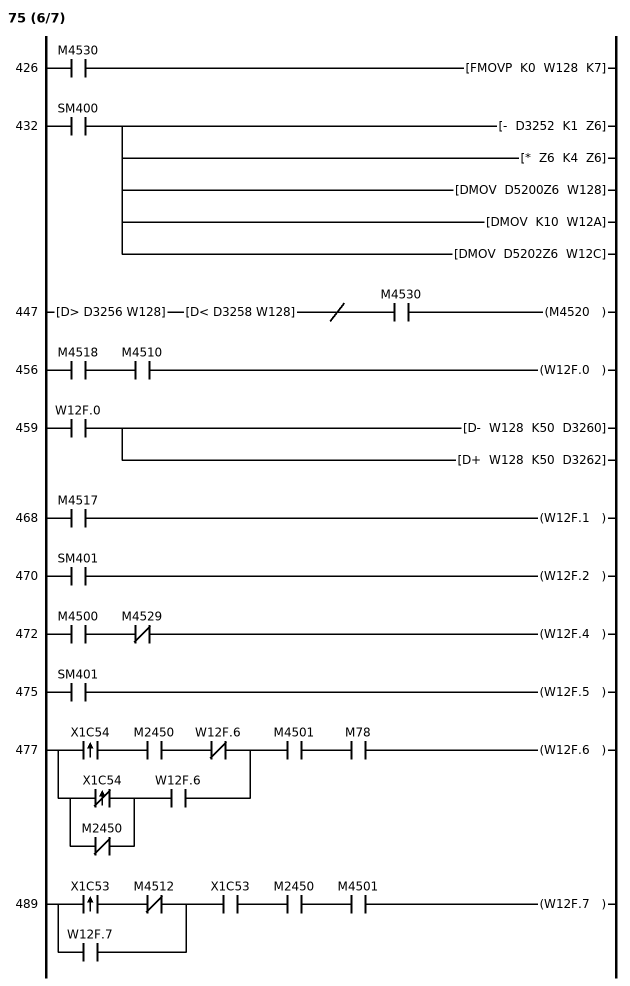
426   LD      M4530
      FMOVP   K0 W128 K7
432   LD      SM400
      -       D3252 K1 Z6
      *       Z6 K4 Z6
      DMOV    D5200Z6 W128
      DMOV    K10 W12A
      DMOV    D5202Z6 W12C
447   LDD>    D3256 W128
      ANDD<   D3258 W128
      INV
      AND     M4530
      OUT     M4520
456   LD      M4518
      AND     M4510
      OUT     W12F.0
459   LD      W12F.0
      D-      W128 K50 D3260
      D+      W128 K50 D3262
468   LD      M4517
      OUT     W12F.1
470   LD      SM401
      OUT     W12F.2
472   LD      M4500
      ANI     M4529
      OUT     W12F.4
475   LD      SM401
      OUT     W12F.5
477   LDP     X1C54
      AND     M2450
      ANI     W12F.6
      LDPI    X1C54
      ORI     M2450
      AND     W12F.6
      ORB
      AND     M4501
      AND     M78
      OUT     W12F.6
489   LDP     X1C53
      ANI     M4512
      OR      W12F.7
      AND     X1C53
      AND     M2450
      AND     M4501
      OUT     W12F.7
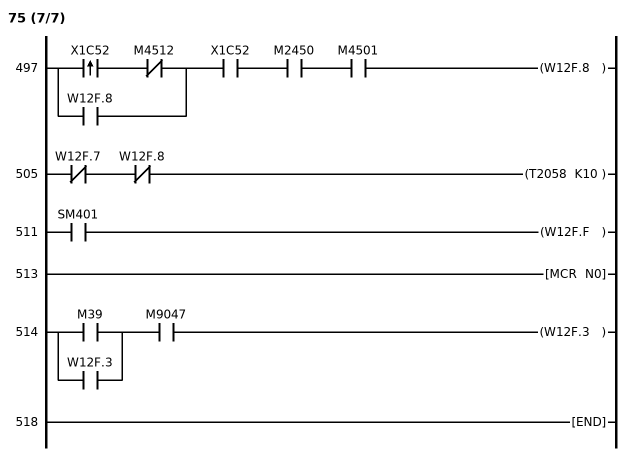
497   LDP     X1C52
      ANI     M4512
      OR      W12F.8
      AND     X1C52
      AND     M2450
      AND     M4501
      OUT     W12F.8
505   LDI     W12F.7
      ANI     W12F.8
      OUT     T2058 K10
511   LD      SM401
      OUT     W12F.F
513   MCR     N0
514   LD      M39
      OR      W12F.3
      AND     M9047
      OUT     W12F.3
518   END
END_PROGRAM

PROGRAM 76
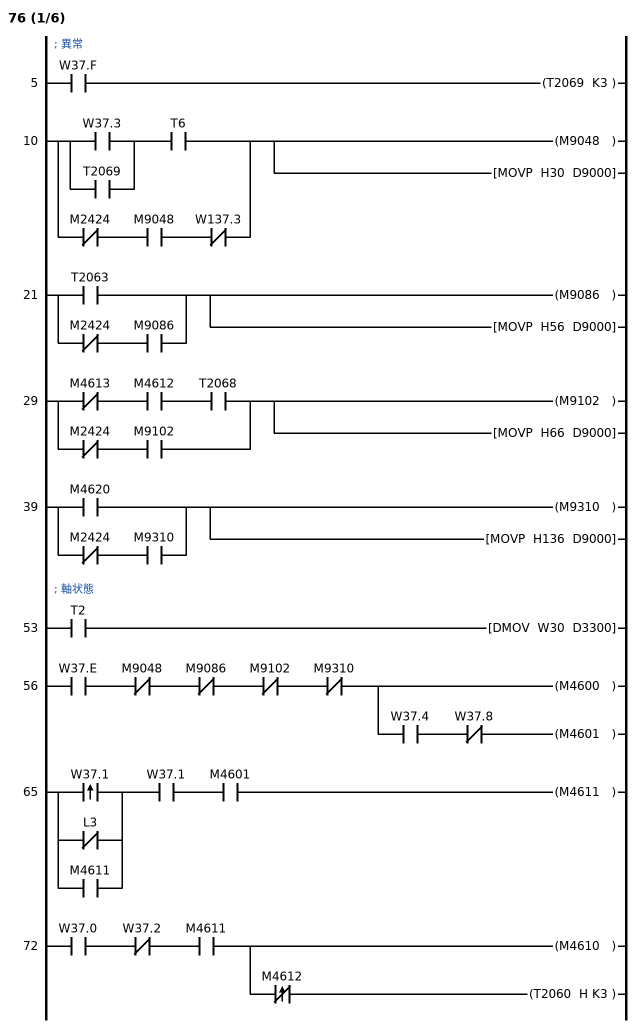
; 異常
5     LD      W37.F
      OUT     T2069 K3
10    LD      W37.3
      OR      T2069
      AND     T6
      LDI     M2424
      AND     M9048
      ANI     W137.3
      ORB
      OUT     M9048
      MOVP    H30 D9000
21    LD      T2063
      LDI     M2424
      AND     M9086
      ORB
      OUT     M9086
      MOVP    H56 D9000
29    LDI     M4613
      AND     M4612
      AND     T2068
      LDI     M2424
      AND     M9102
      ORB
      OUT     M9102
      MOVP    H66 D9000
39    LD      M4620
      LDI     M2424
      AND     M9310
      ORB
      OUT     M9310
      MOVP    H136 D9000
; 軸状態
53    LD      T2
      DMOV    W30 D3300
56    LD      W37.E
      ANI     M9048
      ANI     M9086
      ANI     M9102
      ANI     M9310
      OUT     M4600
      AND     W37.4
      ANI     W37.8
      OUT     M4601
65    LDP     W37.1
      ORI     L3
      OR      M4611
      AND     W37.1
      AND     M4601
      OUT     M4611
72    LD      W37.0
      ANI     W37.2
      AND     M4611
      OUT     M4610
      ANDPI   M4612
      OUTH    T2060 K3
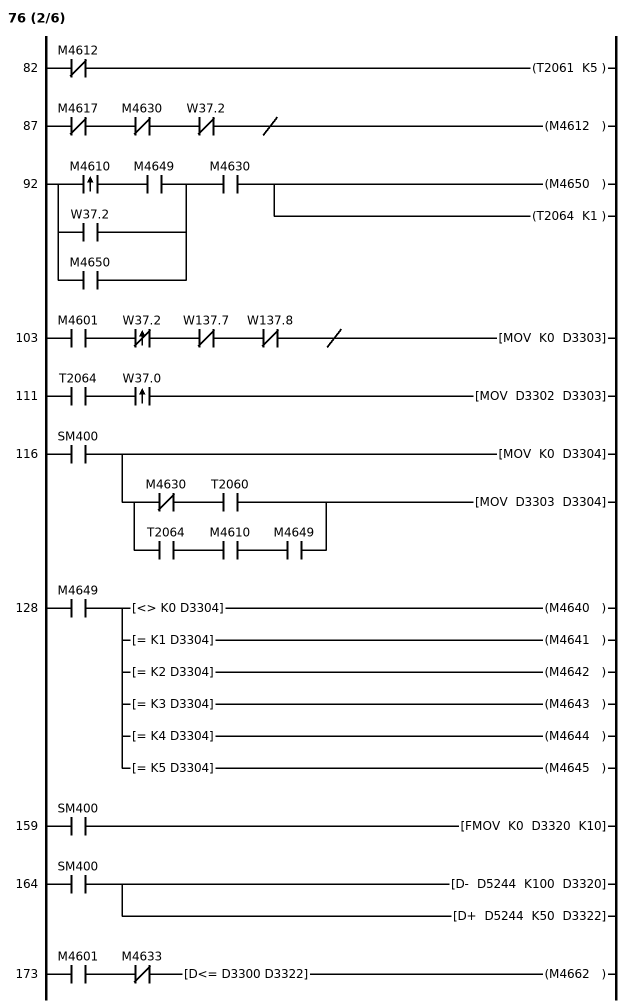
82    LDI     M4612
      OUT     T2061 K5
87    LDI     M4617
      ANI     M4630
      ANI     W37.2
      INV
      OUT     M4612
92    LDP     M4610
      AND     M4649
      OR      W37.2
      OR      M4650
      AND     M4630
      OUT     M4650
      OUT     T2064 K1
103   LD      M4601
      ANDPI   W37.2
      ANI     W137.7
      ANI     W137.8
      INV
      MOV     K0 D3303
111   LD      T2064
      ANDP    W37.0
      MOV     D3302 D3303
116   LD      SM400
      MOV     K0 D3304
      LDI     M4630
      AND     T2060
      LD      T2064
      AND     M4610
      AND     M4649
      ORB
      ANB
      MOV     D3303 D3304
128   LD      M4649
      MPS
      AND<>   K0 D3304
      OUT     M4640
      MRD
      AND=    K1 D3304
      OUT     M4641
      MRD
      AND=    K2 D3304
      OUT     M4642
      MRD
      AND=    K3 D3304
      OUT     M4643
      MRD
      AND=    K4 D3304
      OUT     M4644
      MPP
      AND=    K5 D3304
      OUT     M4645
159   LD      SM400
      FMOV    K0 D3320 K10
164   LD      SM400
      D-      D5244 K100 D3320
      D+      D5244 K50 D3322
173   LD      M4601
      ANI     M4633
      ANDD<=  D3300 D3322
      OUT     M4662
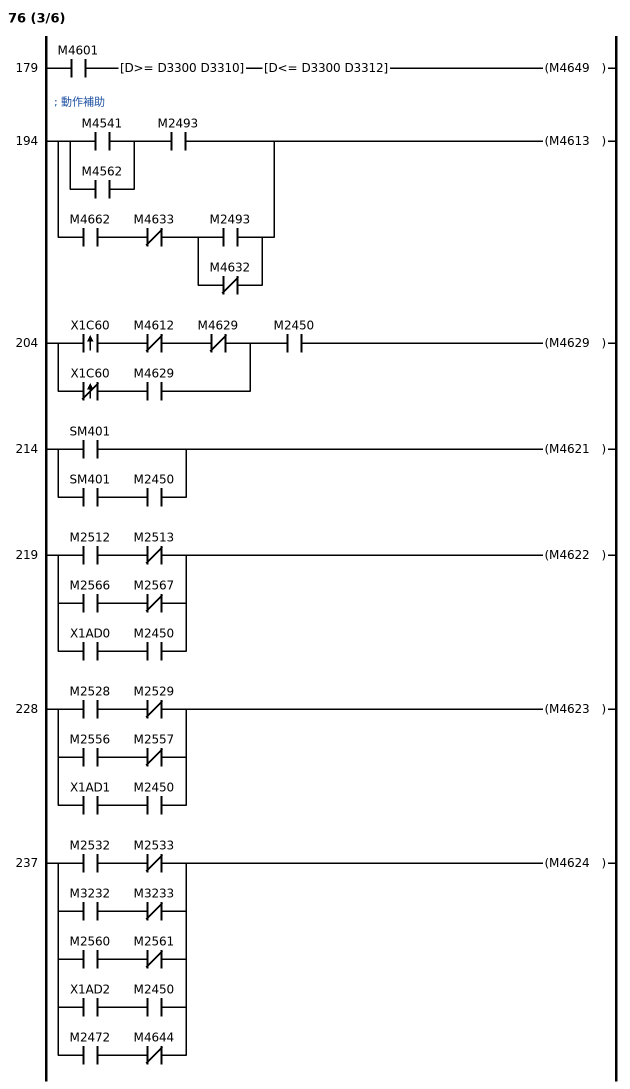
179   LD      M4601
      ANDD>=  D3300 D3310
      ANDD<=  D3300 D3312
      OUT     M4649
; 動作補助
194   LD      M4541
      OR      M4562
      AND     M2493
      LD      M4662
      ANI     M4633
      LD      M2493
      ORI     M4632
      ANB
      ORB
      OUT     M4613
204   LDP     X1C60
      ANI     M4612
      ANI     M4629
      LDPI    X1C60
      AND     M4629
      ORB
      AND     M2450
      OUT     M4629
214   LD      SM401
      LD      SM401
      AND     M2450
      ORB
      OUT     M4621
219   LD      M2512
      ANI     M2513
      LD      M2566
      ANI     M2567
      ORB
      LD      X1AD0
      AND     M2450
      ORB
      OUT     M4622
228   LD      M2528
      ANI     M2529
      LD      M2556
      ANI     M2557
      ORB
      LD      X1AD1
      AND     M2450
      ORB
      OUT     M4623
237   LD      M2532
      ANI     M2533
      LD      M3232
      ANI     M3233
      ORB
      LD      M2560
      ANI     M2561
      ORB
      LD      X1AD2
      AND     M2450
      ORB
      LD      M2472
      ANI     M4644
      ORB
      OUT     M4624
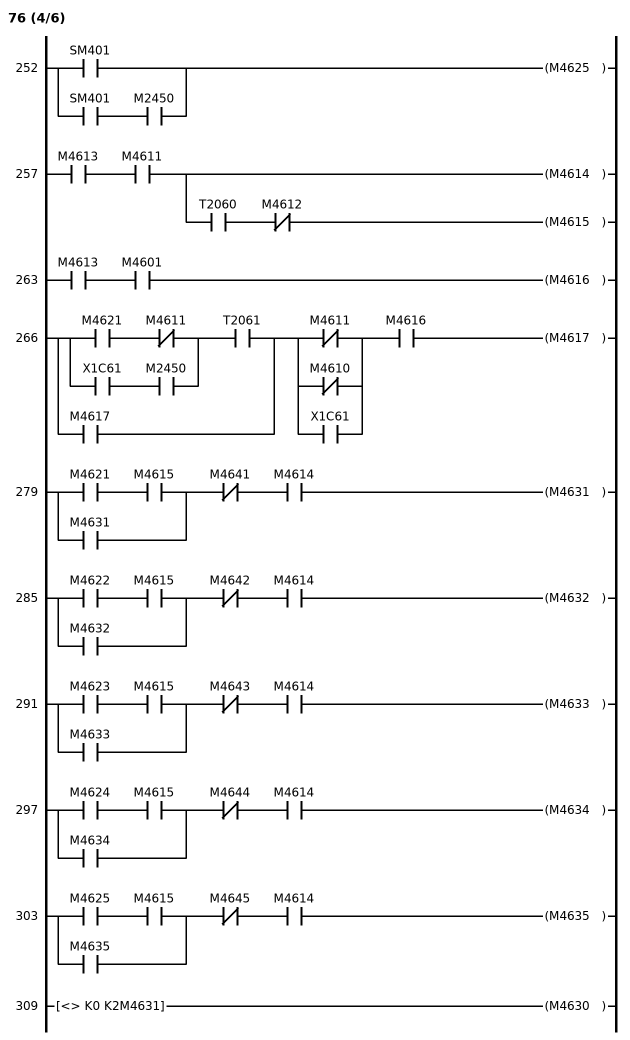
252   LD      SM401
      LD      SM401
      AND     M2450
      ORB
      OUT     M4625
257   LD      M4613
      AND     M4611
      OUT     M4614
      AND     T2060
      ANI     M4612
      OUT     M4615
263   LD      M4613
      AND     M4601
      OUT     M4616
266   LD      M4621
      ANI     M4611
      LD      X1C61
      AND     M2450
      ORB
      AND     T2061
      OR      M4617
      LDI     M4611
      ORI     M4610
      OR      X1C61
      ANB
      AND     M4616
      OUT     M4617
279   LD      M4621
      AND     M4615
      OR      M4631
      ANI     M4641
      AND     M4614
      OUT     M4631
285   LD      M4622
      AND     M4615
      OR      M4632
      ANI     M4642
      AND     M4614
      OUT     M4632
291   LD      M4623
      AND     M4615
      OR      M4633
      ANI     M4643
      AND     M4614
      OUT     M4633
297   LD      M4624
      AND     M4615
      OR      M4634
      ANI     M4644
      AND     M4614
      OUT     M4634
303   LD      M4625
      AND     M4615
      OR      M4635
      ANI     M4645
      AND     M4614
      OUT     M4635
309   LD<>    K0 K2M4631
      OUT     M4630
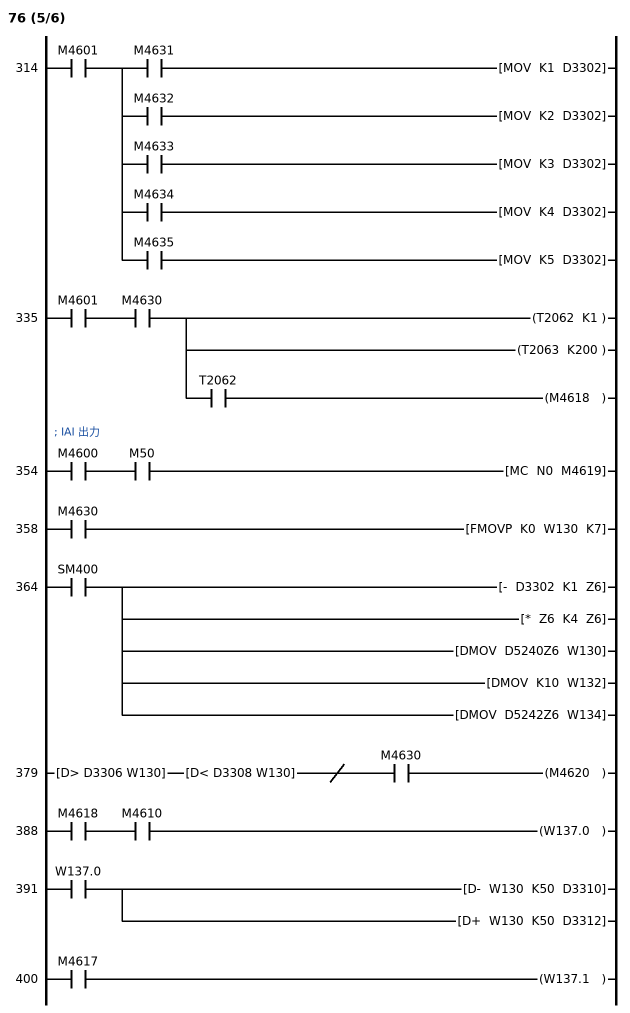
314   LD      M4601
      MPS
      AND     M4631
      MOV     K1 D3302
      MRD
      AND     M4632
      MOV     K2 D3302
      MRD
      AND     M4633
      MOV     K3 D3302
      MRD
      AND     M4634
      MOV     K4 D3302
      MPP
      AND     M4635
      MOV     K5 D3302
335   LD      M4601
      AND     M4630
      OUT     T2062 K1
      OUT     T2063 K200
      AND     T2062
      OUT     M4618
; IAI 出力
354   LD      M4600
      AND     M50
      MC      N0 M4619
358   LD      M4630
      FMOVP   K0 W130 K7
364   LD      SM400
      -       D3302 K1 Z6
      *       Z6 K4 Z6
      DMOV    D5240Z6 W130
      DMOV    K10 W132
      DMOV    D5242Z6 W134
379   LDD>    D3306 W130
      ANDD<   D3308 W130
      INV
      AND     M4630
      OUT     M4620
388   LD      M4618
      AND     M4610
      OUT     W137.0
391   LD      W137.0
      D-      W130 K50 D3310
      D+      W130 K50 D3312
400   LD      M4617
      OUT     W137.1
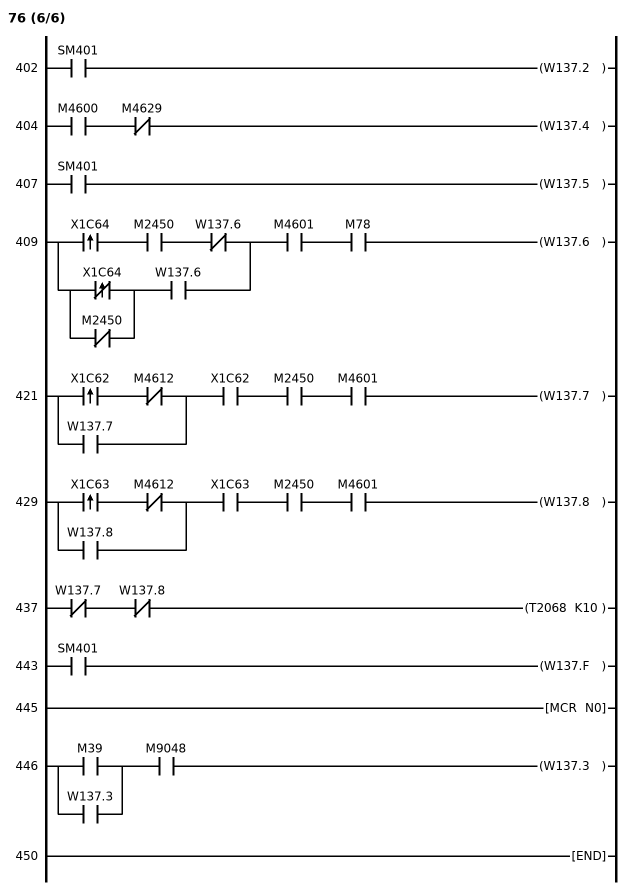
402   LD      SM401
      OUT     W137.2
404   LD      M4600
      ANI     M4629
      OUT     W137.4
407   LD      SM401
      OUT     W137.5
409   LDP     X1C64
      AND     M2450
      ANI     W137.6
      LDPI    X1C64
      ORI     M2450
      AND     W137.6
      ORB
      AND     M4601
      AND     M78
      OUT     W137.6
421   LDP     X1C62
      ANI     M4612
      OR      W137.7
      AND     X1C62
      AND     M2450
      AND     M4601
      OUT     W137.7
429   LDP     X1C63
      ANI     M4612
      OR      W137.8
      AND     X1C63
      AND     M2450
      AND     M4601
      OUT     W137.8
437   LDI     W137.7
      ANI     W137.8
      OUT     T2068 K10
443   LD      SM401
      OUT     W137.F
445   MCR     N0
446   LD      M39
      OR      W137.3
      AND     M9048
      OUT     W137.3
450   END
END_PROGRAM

PROGRAM 77
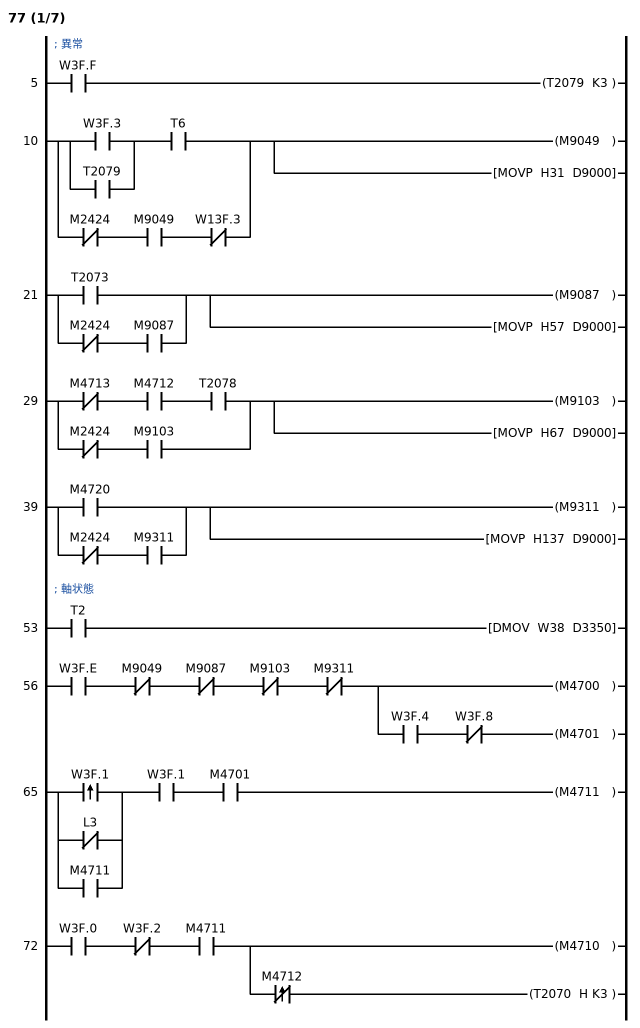
; 異常
5     LD      W3F.F
      OUT     T2079 K3
10    LD      W3F.3
      OR      T2079
      AND     T6
      LDI     M2424
      AND     M9049
      ANI     W13F.3
      ORB
      OUT     M9049
      MOVP    H31 D9000
21    LD      T2073
      LDI     M2424
      AND     M9087
      ORB
      OUT     M9087
      MOVP    H57 D9000
29    LDI     M4713
      AND     M4712
      AND     T2078
      LDI     M2424
      AND     M9103
      ORB
      OUT     M9103
      MOVP    H67 D9000
39    LD      M4720
      LDI     M2424
      AND     M9311
      ORB
      OUT     M9311
      MOVP    H137 D9000
; 軸状態
53    LD      T2
      DMOV    W38 D3350
56    LD      W3F.E
      ANI     M9049
      ANI     M9087
      ANI     M9103
      ANI     M9311
      OUT     M4700
      AND     W3F.4
      ANI     W3F.8
      OUT     M4701
65    LDP     W3F.1
      ORI     L3
      OR      M4711
      AND     W3F.1
      AND     M4701
      OUT     M4711
72    LD      W3F.0
      ANI     W3F.2
      AND     M4711
      OUT     M4710
      ANDPI   M4712
      OUTH    T2070 K3
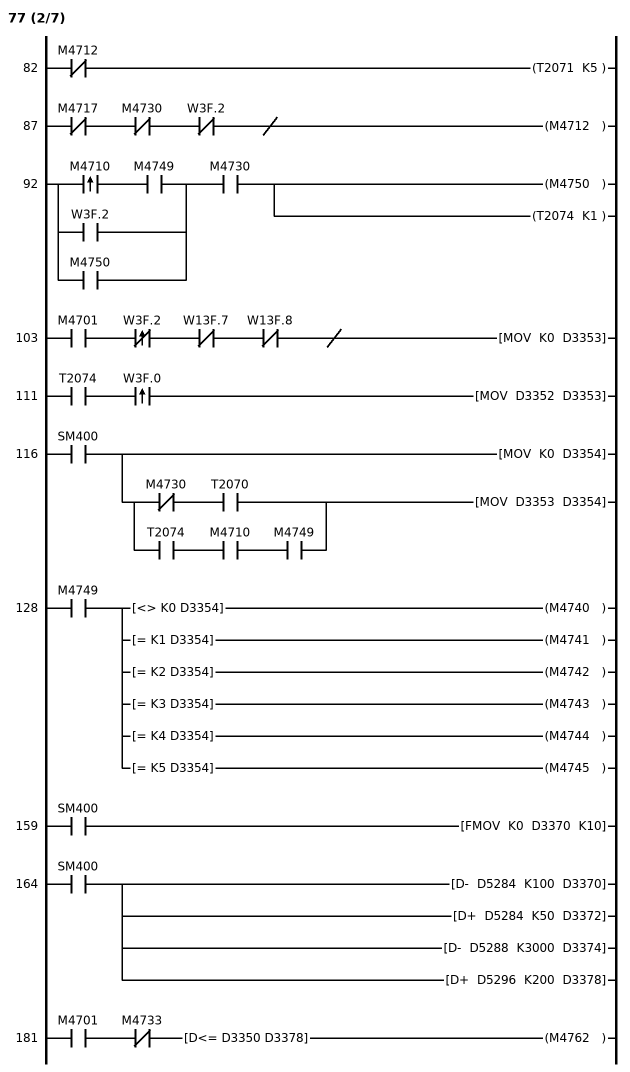
82    LDI     M4712
      OUT     T2071 K5
87    LDI     M4717
      ANI     M4730
      ANI     W3F.2
      INV
      OUT     M4712
92    LDP     M4710
      AND     M4749
      OR      W3F.2
      OR      M4750
      AND     M4730
      OUT     M4750
      OUT     T2074 K1
103   LD      M4701
      ANDPI   W3F.2
      ANI     W13F.7
      ANI     W13F.8
      INV
      MOV     K0 D3353
111   LD      T2074
      ANDP    W3F.0
      MOV     D3352 D3353
116   LD      SM400
      MOV     K0 D3354
      LDI     M4730
      AND     T2070
      LD      T2074
      AND     M4710
      AND     M4749
      ORB
      ANB
      MOV     D3353 D3354
128   LD      M4749
      MPS
      AND<>   K0 D3354
      OUT     M4740
      MRD
      AND=    K1 D3354
      OUT     M4741
      MRD
      AND=    K2 D3354
      OUT     M4742
      MRD
      AND=    K3 D3354
      OUT     M4743
      MRD
      AND=    K4 D3354
      OUT     M4744
      MPP
      AND=    K5 D3354
      OUT     M4745
159   LD      SM400
      FMOV    K0 D3370 K10
164   LD      SM400
      D-      D5284 K100 D3370
      D+      D5284 K50 D3372
      D-      D5288 K3000 D3374
      D+      D5296 K200 D3378
181   LD      M4701
      ANI     M4733
      ANDD<=  D3350 D3378
      OUT     M4762
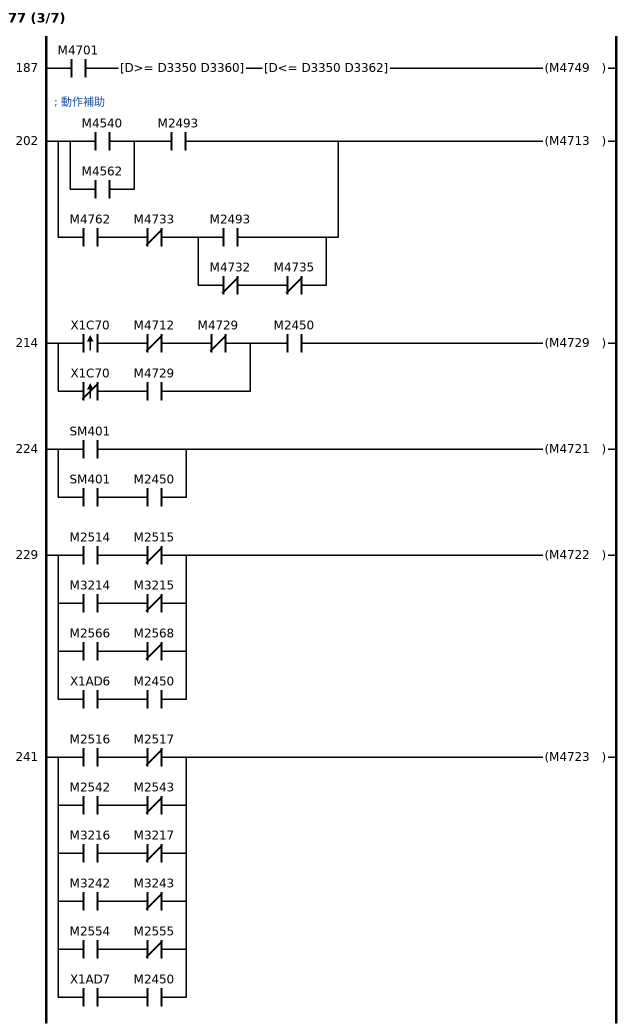
187   LD      M4701
      ANDD>=  D3350 D3360
      ANDD<=  D3350 D3362
      OUT     M4749
; 動作補助
202   LD      M4540
      OR      M4562
      AND     M2493
      LD      M4762
      ANI     M4733
      LD      M2493
      LDI     M4732
      ANI     M4735
      ORB
      ANB
      ORB
      OUT     M4713
214   LDP     X1C70
      ANI     M4712
      ANI     M4729
      LDPI    X1C70
      AND     M4729
      ORB
      AND     M2450
      OUT     M4729
224   LD      SM401
      LD      SM401
      AND     M2450
      ORB
      OUT     M4721
229   LD      M2514
      ANI     M2515
      LD      M3214
      ANI     M3215
      ORB
      LD      M2566
      ANI     M2568
      ORB
      LD      X1AD6
      AND     M2450
      ORB
      OUT     M4722
241   LD      M2516
      ANI     M2517
      LD      M2542
      ANI     M2543
      ORB
      LD      M3216
      ANI     M3217
      ORB
      LD      M3242
      ANI     M3243
      ORB
      LD      M2554
      ANI     M2555
      ORB
      LD      X1AD7
      AND     M2450
      ORB
      OUT     M4723
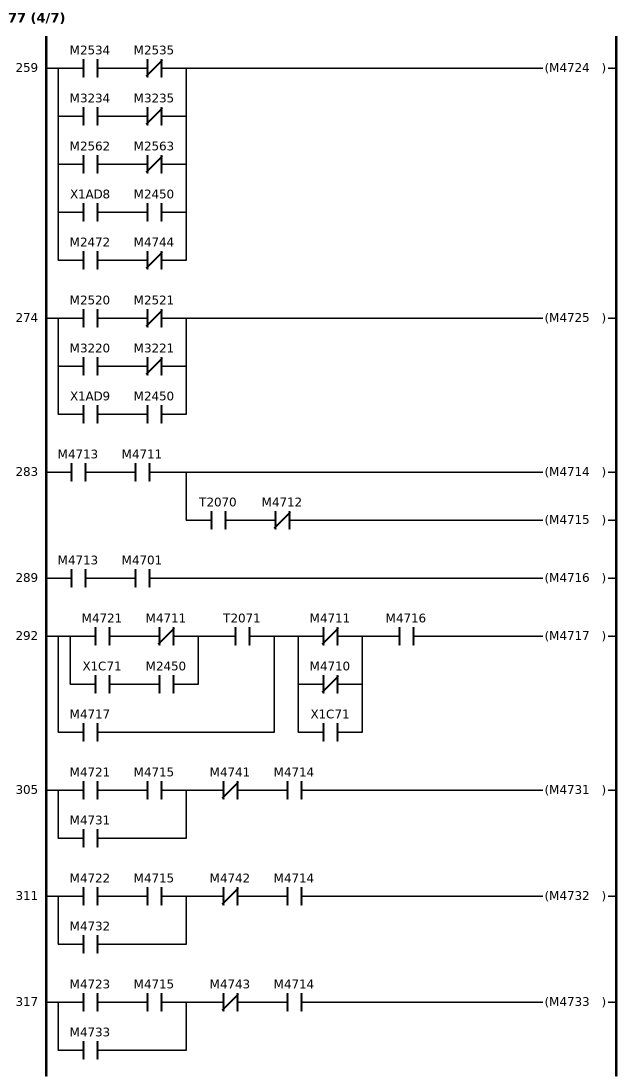
259   LD      M2534
      ANI     M2535
      LD      M3234
      ANI     M3235
      ORB
      LD      M2562
      ANI     M2563
      ORB
      LD      X1AD8
      AND     M2450
      ORB
      LD      M2472
      ANI     M4744
      ORB
      OUT     M4724
274   LD      M2520
      ANI     M2521
      LD      M3220
      ANI     M3221
      ORB
      LD      X1AD9
      AND     M2450
      ORB
      OUT     M4725
283   LD      M4713
      AND     M4711
      OUT     M4714
      AND     T2070
      ANI     M4712
      OUT     M4715
289   LD      M4713
      AND     M4701
      OUT     M4716
292   LD      M4721
      ANI     M4711
      LD      X1C71
      AND     M2450
      ORB
      AND     T2071
      OR      M4717
      LDI     M4711
      ORI     M4710
      OR      X1C71
      ANB
      AND     M4716
      OUT     M4717
305   LD      M4721
      AND     M4715
      OR      M4731
      ANI     M4741
      AND     M4714
      OUT     M4731
311   LD      M4722
      AND     M4715
      OR      M4732
      ANI     M4742
      AND     M4714
      OUT     M4732
317   LD      M4723
      AND     M4715
      OR      M4733
      ANI     M4743
      AND     M4714
      OUT     M4733
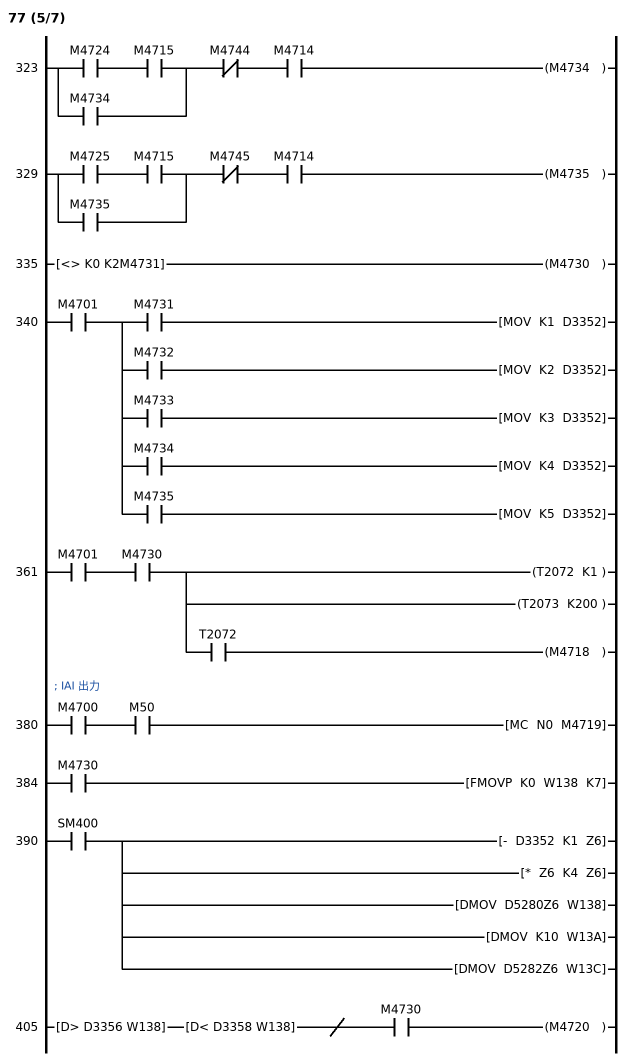
323   LD      M4724
      AND     M4715
      OR      M4734
      ANI     M4744
      AND     M4714
      OUT     M4734
329   LD      M4725
      AND     M4715
      OR      M4735
      ANI     M4745
      AND     M4714
      OUT     M4735
335   LD<>    K0 K2M4731
      OUT     M4730
340   LD      M4701
      MPS
      AND     M4731
      MOV     K1 D3352
      MRD
      AND     M4732
      MOV     K2 D3352
      MRD
      AND     M4733
      MOV     K3 D3352
      MRD
      AND     M4734
      MOV     K4 D3352
      MPP
      AND     M4735
      MOV     K5 D3352
361   LD      M4701
      AND     M4730
      OUT     T2072 K1
      OUT     T2073 K200
      AND     T2072
      OUT     M4718
; IAI 出力
380   LD      M4700
      AND     M50
      MC      N0 M4719
384   LD      M4730
      FMOVP   K0 W138 K7
390   LD      SM400
      -       D3352 K1 Z6
      *       Z6 K4 Z6
      DMOV    D5280Z6 W138
      DMOV    K10 W13A
      DMOV    D5282Z6 W13C
405   LDD>    D3356 W138
      ANDD<   D3358 W138
      INV
      AND     M4730
      OUT     M4720
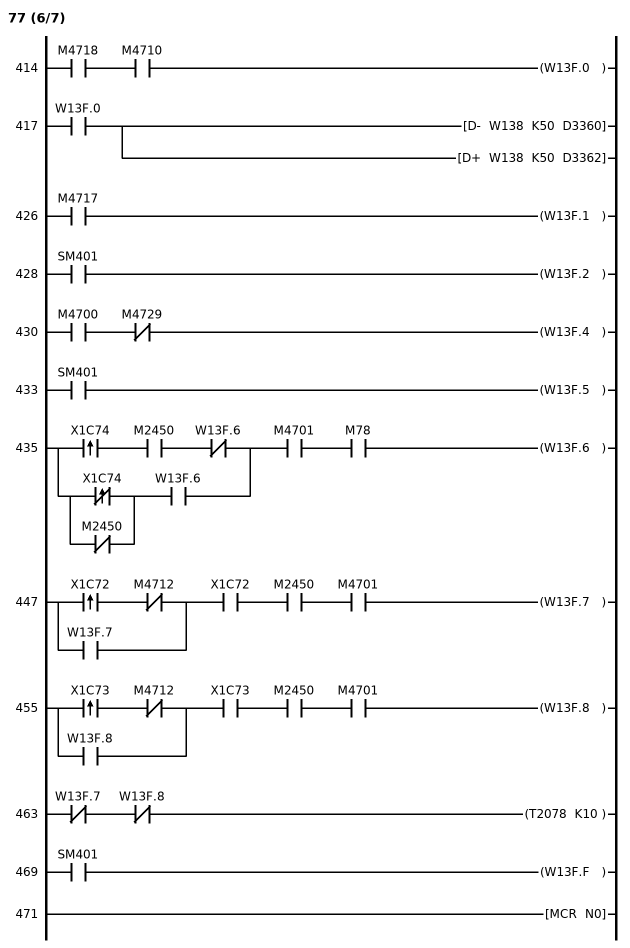
414   LD      M4718
      AND     M4710
      OUT     W13F.0
417   LD      W13F.0
      D-      W138 K50 D3360
      D+      W138 K50 D3362
426   LD      M4717
      OUT     W13F.1
428   LD      SM401
      OUT     W13F.2
430   LD      M4700
      ANI     M4729
      OUT     W13F.4
433   LD      SM401
      OUT     W13F.5
435   LDP     X1C74
      AND     M2450
      ANI     W13F.6
      LDPI    X1C74
      ORI     M2450
      AND     W13F.6
      ORB
      AND     M4701
      AND     M78
      OUT     W13F.6
447   LDP     X1C72
      ANI     M4712
      OR      W13F.7
      AND     X1C72
      AND     M2450
      AND     M4701
      OUT     W13F.7
455   LDP     X1C73
      ANI     M4712
      OR      W13F.8
      AND     X1C73
      AND     M2450
      AND     M4701
      OUT     W13F.8
463   LDI     W13F.7
      ANI     W13F.8
      OUT     T2078 K10
469   LD      SM401
      OUT     W13F.F
471   MCR     N0
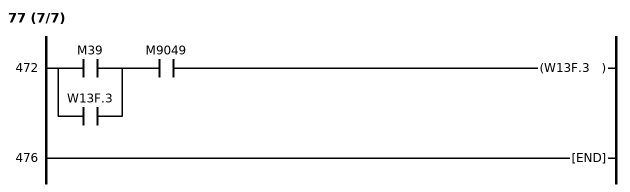
472   LD      M39
      OR      W13F.3
      AND     M9049
      OUT     W13F.3
476   END
END_PROGRAM

PROGRAM 78
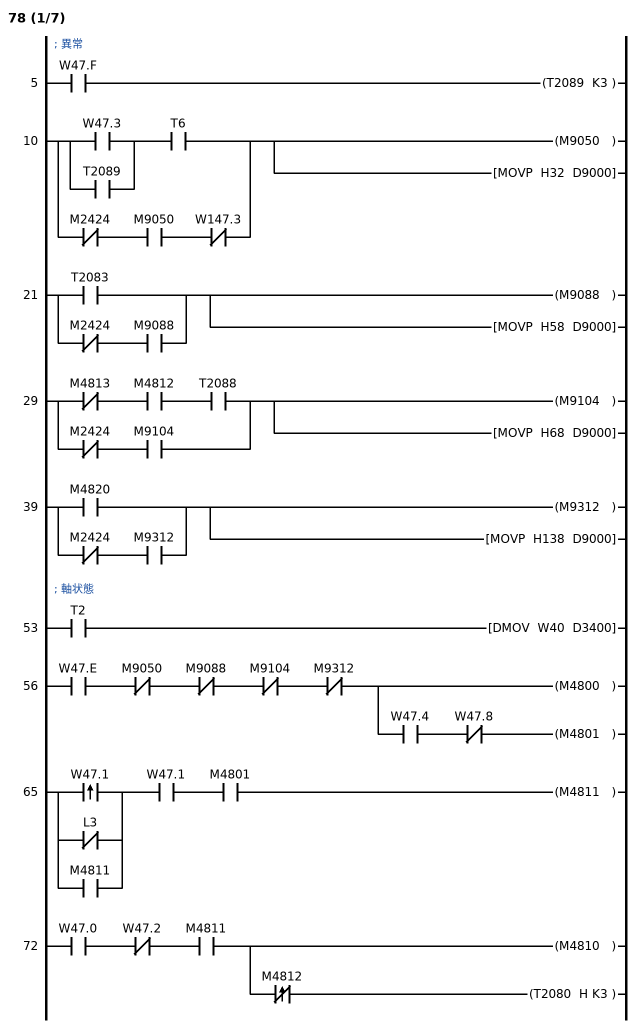
; 異常
5     LD      W47.F
      OUT     T2089 K3
10    LD      W47.3
      OR      T2089
      AND     T6
      LDI     M2424
      AND     M9050
      ANI     W147.3
      ORB
      OUT     M9050
      MOVP    H32 D9000
21    LD      T2083
      LDI     M2424
      AND     M9088
      ORB
      OUT     M9088
      MOVP    H58 D9000
29    LDI     M4813
      AND     M4812
      AND     T2088
      LDI     M2424
      AND     M9104
      ORB
      OUT     M9104
      MOVP    H68 D9000
39    LD      M4820
      LDI     M2424
      AND     M9312
      ORB
      OUT     M9312
      MOVP    H138 D9000
; 軸状態
53    LD      T2
      DMOV    W40 D3400
56    LD      W47.E
      ANI     M9050
      ANI     M9088
      ANI     M9104
      ANI     M9312
      OUT     M4800
      AND     W47.4
      ANI     W47.8
      OUT     M4801
65    LDP     W47.1
      ORI     L3
      OR      M4811
      AND     W47.1
      AND     M4801
      OUT     M4811
72    LD      W47.0
      ANI     W47.2
      AND     M4811
      OUT     M4810
      ANDPI   M4812
      OUTH    T2080 K3
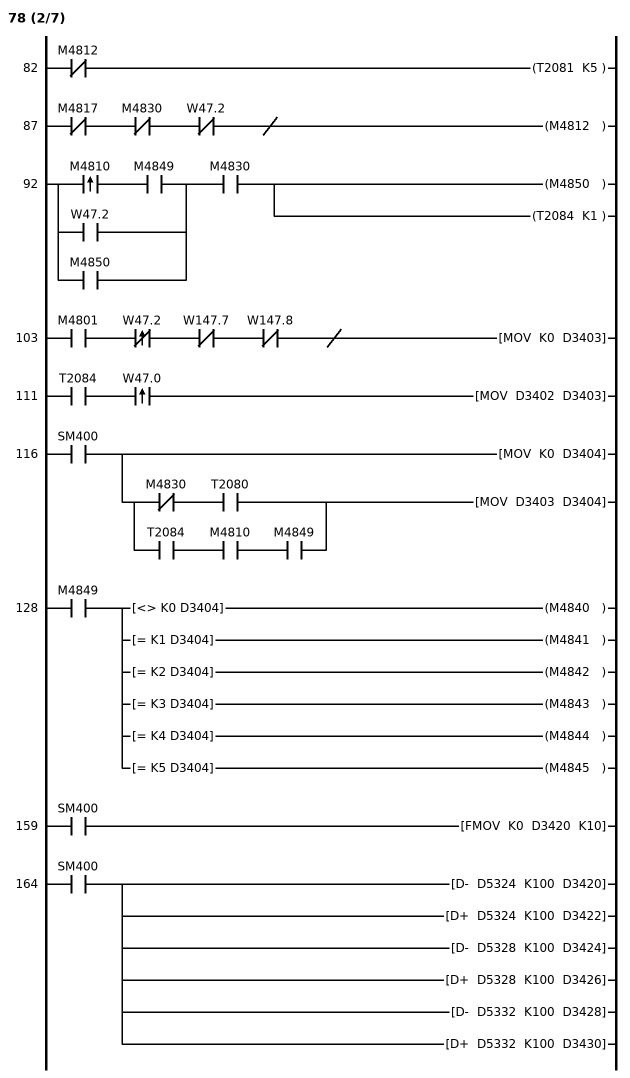
82    LDI     M4812
      OUT     T2081 K5
87    LDI     M4817
      ANI     M4830
      ANI     W47.2
      INV
      OUT     M4812
92    LDP     M4810
      AND     M4849
      OR      W47.2
      OR      M4850
      AND     M4830
      OUT     M4850
      OUT     T2084 K1
103   LD      M4801
      ANDPI   W47.2
      ANI     W147.7
      ANI     W147.8
      INV
      MOV     K0 D3403
111   LD      T2084
      ANDP    W47.0
      MOV     D3402 D3403
116   LD      SM400
      MOV     K0 D3404
      LDI     M4830
      AND     T2080
      LD      T2084
      AND     M4810
      AND     M4849
      ORB
      ANB
      MOV     D3403 D3404
128   LD      M4849
      MPS
      AND<>   K0 D3404
      OUT     M4840
      MRD
      AND=    K1 D3404
      OUT     M4841
      MRD
      AND=    K2 D3404
      OUT     M4842
      MRD
      AND=    K3 D3404
      OUT     M4843
      MRD
      AND=    K4 D3404
      OUT     M4844
      MPP
      AND=    K5 D3404
      OUT     M4845
159   LD      SM400
      FMOV    K0 D3420 K10
164   LD      SM400
      D-      D5324 K100 D3420
      D+      D5324 K100 D3422
      D-      D5328 K100 D3424
      D+      D5328 K100 D3426
      D-      D5332 K100 D3428
      D+      D5332 K100 D3430
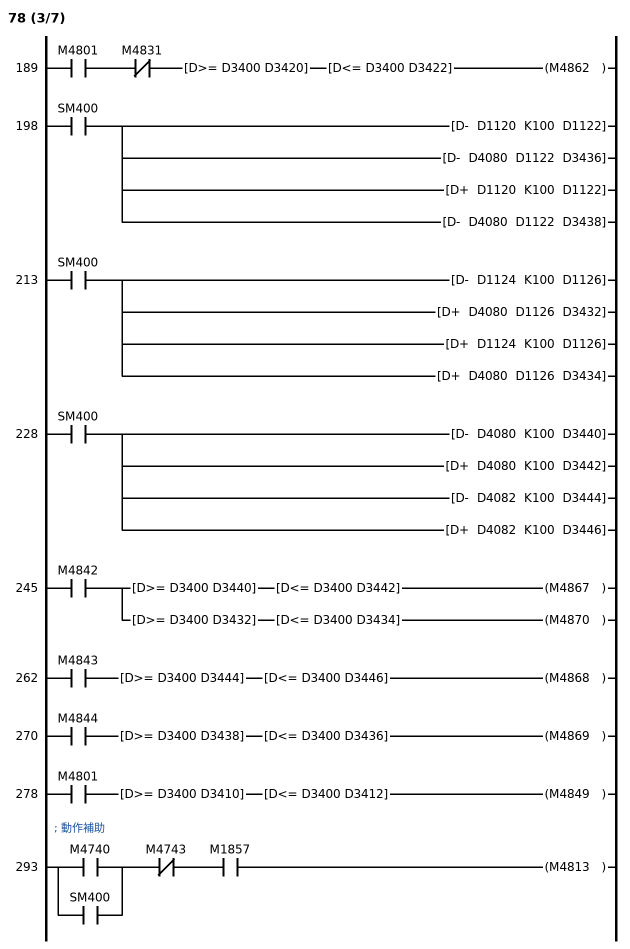
189   LD      M4801
      ANI     M4831
      ANDD>=  D3400 D3420
      ANDD<=  D3400 D3422
      OUT     M4862
198   LD      SM400
      D-      D1120 K100 D1122
      D-      D4080 D1122 D3436
      D+      D1120 K100 D1122
      D-      D4080 D1122 D3438
213   LD      SM400
      D-      D1124 K100 D1126
      D+      D4080 D1126 D3432
      D+      D1124 K100 D1126
      D+      D4080 D1126 D3434
228   LD      SM400
      D-      D4080 K100 D3440
      D+      D4080 K100 D3442
      D-      D4082 K100 D3444
      D+      D4082 K100 D3446
245   LD      M4842
      MPS
      ANDD>=  D3400 D3440
      ANDD<=  D3400 D3442
      OUT     M4867
      MPP
      ANDD>=  D3400 D3432
      ANDD<=  D3400 D3434
      OUT     M4870
262   LD      M4843
      ANDD>=  D3400 D3444
      ANDD<=  D3400 D3446
      OUT     M4868
270   LD      M4844
      ANDD>=  D3400 D3438
      ANDD<=  D3400 D3436
      OUT     M4869
278   LD      M4801
      ANDD>=  D3400 D3410
      ANDD<=  D3400 D3412
      OUT     M4849
; 動作補助
293   LD      M4740
      OR      SM400
      ANI     M4743
      AND     M1857
      OUT     M4813
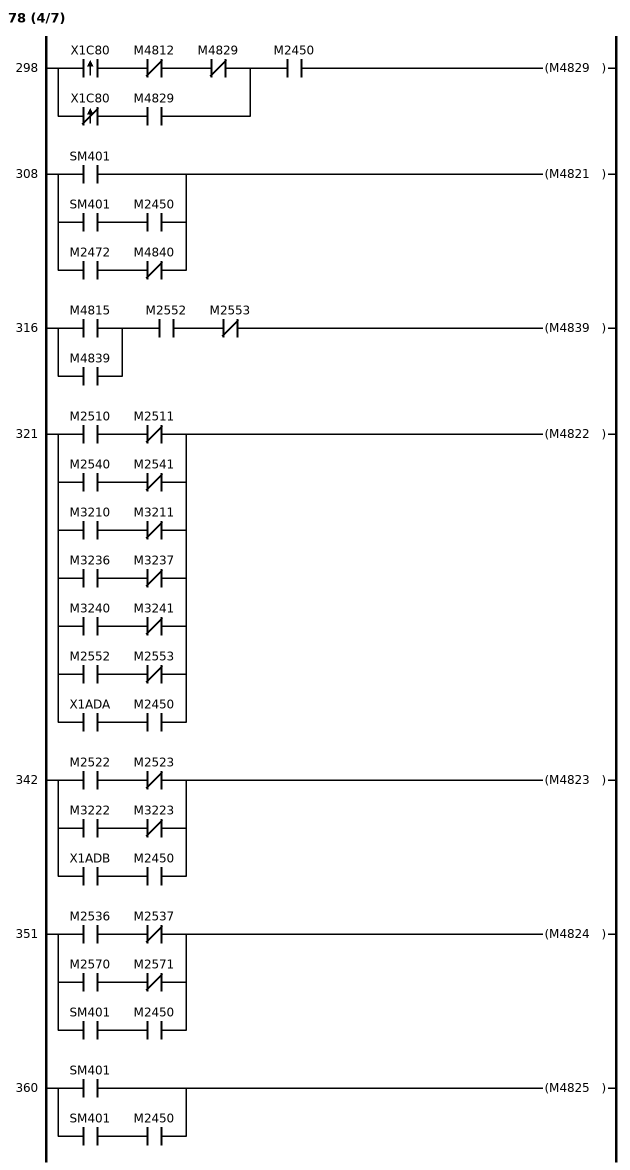
298   LDP     X1C80
      ANI     M4812
      ANI     M4829
      LDPI    X1C80
      AND     M4829
      ORB
      AND     M2450
      OUT     M4829
308   LD      SM401
      LD      SM401
      AND     M2450
      ORB
      LD      M2472
      ANI     M4840
      ORB
      OUT     M4821
316   LD      M4815
      OR      M4839
      AND     M2552
      ANI     M2553
      OUT     M4839
321   LD      M2510
      ANI     M2511
      LD      M2540
      ANI     M2541
      ORB
      LD      M3210
      ANI     M3211
      ORB
      LD      M3236
      ANI     M3237
      ORB
      LD      M3240
      ANI     M3241
      ORB
      LD      M2552
      ANI     M2553
      ORB
      LD      X1ADA
      AND     M2450
      ORB
      OUT     M4822
342   LD      M2522
      ANI     M2523
      LD      M3222
      ANI     M3223
      ORB
      LD      X1ADB
      AND     M2450
      ORB
      OUT     M4823
351   LD      M2536
      ANI     M2537
      LD      M2570
      ANI     M2571
      ORB
      LD      SM401
      AND     M2450
      ORB
      OUT     M4824
360   LD      SM401
      LD      SM401
      AND     M2450
      ORB
      OUT     M4825
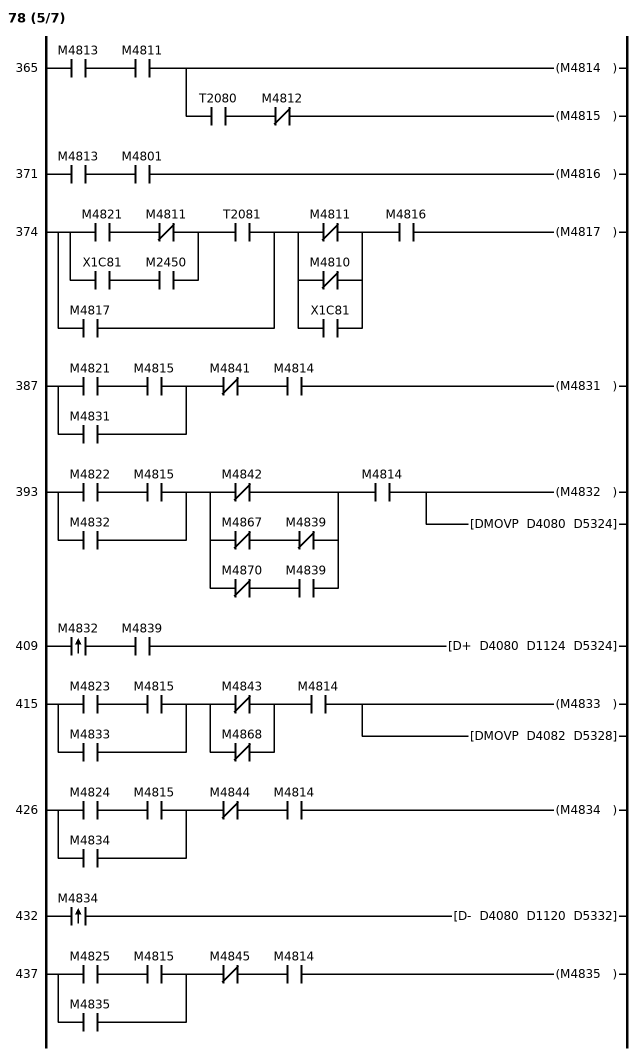
365   LD      M4813
      AND     M4811
      OUT     M4814
      AND     T2080
      ANI     M4812
      OUT     M4815
371   LD      M4813
      AND     M4801
      OUT     M4816
374   LD      M4821
      ANI     M4811
      LD      X1C81
      AND     M2450
      ORB
      AND     T2081
      OR      M4817
      LDI     M4811
      ORI     M4810
      OR      X1C81
      ANB
      AND     M4816
      OUT     M4817
387   LD      M4821
      AND     M4815
      OR      M4831
      ANI     M4841
      AND     M4814
      OUT     M4831
393   LD      M4822
      AND     M4815
      OR      M4832
      LDI     M4842
      LDI     M4867
      ANI     M4839
      ORB
      LDI     M4870
      AND     M4839
      ORB
      ANB
      AND     M4814
      OUT     M4832
      DMOVP   D4080 D5324
409   LDP     M4832
      AND     M4839
      D+      D4080 D1124 D5324
415   LD      M4823
      AND     M4815
      OR      M4833
      LDI     M4843
      ORI     M4868
      ANB
      AND     M4814
      OUT     M4833
      DMOVP   D4082 D5328
426   LD      M4824
      AND     M4815
      OR      M4834
      ANI     M4844
      AND     M4814
      OUT     M4834
432   LDP     M4834
      D-      D4080 D1120 D5332
437   LD      M4825
      AND     M4815
      OR      M4835
      ANI     M4845
      AND     M4814
      OUT     M4835
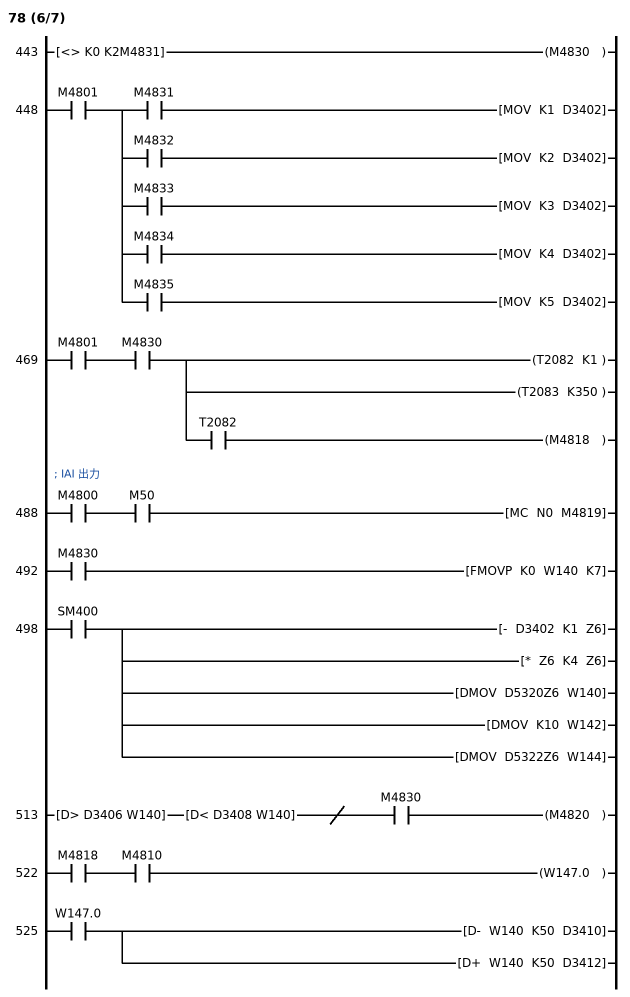
443   LD<>    K0 K2M4831
      OUT     M4830
448   LD      M4801
      MPS
      AND     M4831
      MOV     K1 D3402
      MRD
      AND     M4832
      MOV     K2 D3402
      MRD
      AND     M4833
      MOV     K3 D3402
      MRD
      AND     M4834
      MOV     K4 D3402
      MPP
      AND     M4835
      MOV     K5 D3402
469   LD      M4801
      AND     M4830
      OUT     T2082 K1
      OUT     T2083 K350
      AND     T2082
      OUT     M4818
; IAI 出力
488   LD      M4800
      AND     M50
      MC      N0 M4819
492   LD      M4830
      FMOVP   K0 W140 K7
498   LD      SM400
      -       D3402 K1 Z6
      *       Z6 K4 Z6
      DMOV    D5320Z6 W140
      DMOV    K10 W142
      DMOV    D5322Z6 W144
513   LDD>    D3406 W140
      ANDD<   D3408 W140
      INV
      AND     M4830
      OUT     M4820
522   LD      M4818
      AND     M4810
      OUT     W147.0
525   LD      W147.0
      D-      W140 K50 D3410
      D+      W140 K50 D3412
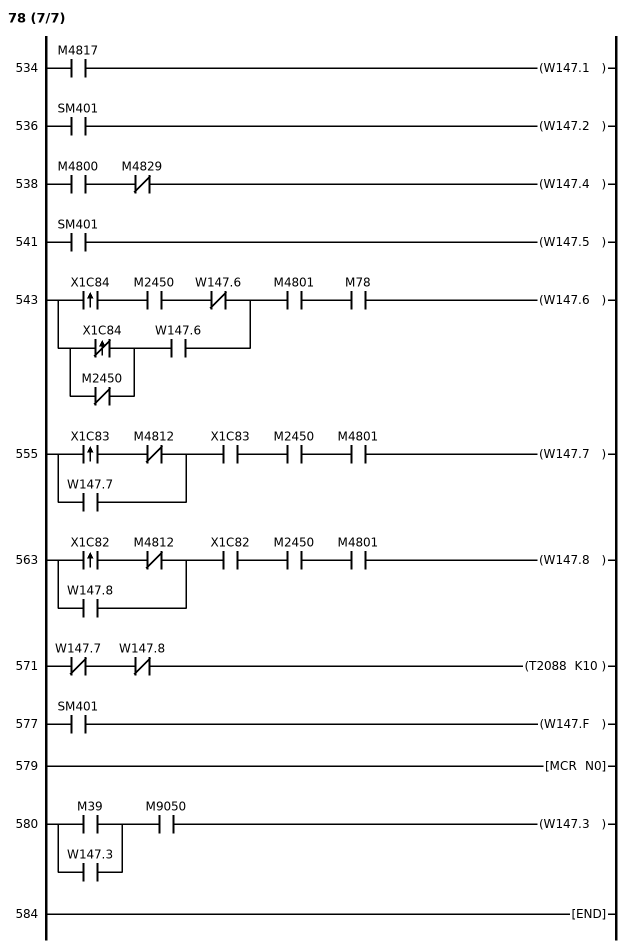
534   LD      M4817
      OUT     W147.1
536   LD      SM401
      OUT     W147.2
538   LD      M4800
      ANI     M4829
      OUT     W147.4
541   LD      SM401
      OUT     W147.5
543   LDP     X1C84
      AND     M2450
      ANI     W147.6
      LDPI    X1C84
      ORI     M2450
      AND     W147.6
      ORB
      AND     M4801
      AND     M78
      OUT     W147.6
555   LDP     X1C83
      ANI     M4812
      OR      W147.7
      AND     X1C83
      AND     M2450
      AND     M4801
      OUT     W147.7
563   LDP     X1C82
      ANI     M4812
      OR      W147.8
      AND     X1C82
      AND     M2450
      AND     M4801
      OUT     W147.8
571   LDI     W147.7
      ANI     W147.8
      OUT     T2088 K10
577   LD      SM401
      OUT     W147.F
579   MCR     N0
580   LD      M39
      OR      W147.3
      AND     M9050
      OUT     W147.3
584   END
END_PROGRAM

PROGRAM 79
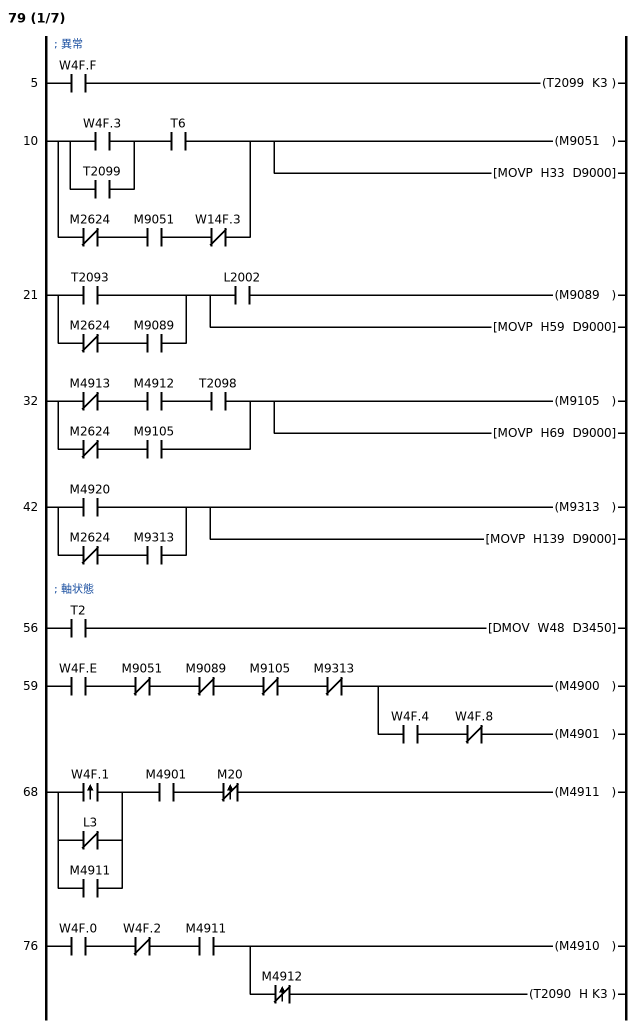
; 異常
5     LD      W4F.F
      OUT     T2099 K3
10    LD      W4F.3
      OR      T2099
      AND     T6
      LDI     M2624
      AND     M9051
      ANI     W14F.3
      ORB
      OUT     M9051
      MOVP    H33 D9000
21    LD      T2093
      LDI     M2624
      AND     M9089
      ORB
      MPS
      AND     L2002
      OUT     M9089
      MPP
      MOVP    H59 D9000
32    LDI     M4913
      AND     M4912
      AND     T2098
      LDI     M2624
      AND     M9105
      ORB
      OUT     M9105
      MOVP    H69 D9000
42    LD      M4920
      LDI     M2624
      AND     M9313
      ORB
      OUT     M9313
      MOVP    H139 D9000
; 軸状態
56    LD      T2
      DMOV    W48 D3450
59    LD      W4F.E
      ANI     M9051
      ANI     M9089
      ANI     M9105
      ANI     M9313
      OUT     M4900
      AND     W4F.4
      ANI     W4F.8
      OUT     M4901
68    LDP     W4F.1
      ORI     L3
      OR      M4911
      AND     M4901
      ANDPI   M20
      OUT     M4911
76    LD      W4F.0
      ANI     W4F.2
      AND     M4911
      OUT     M4910
      ANDPI   M4912
      OUTH    T2090 K3
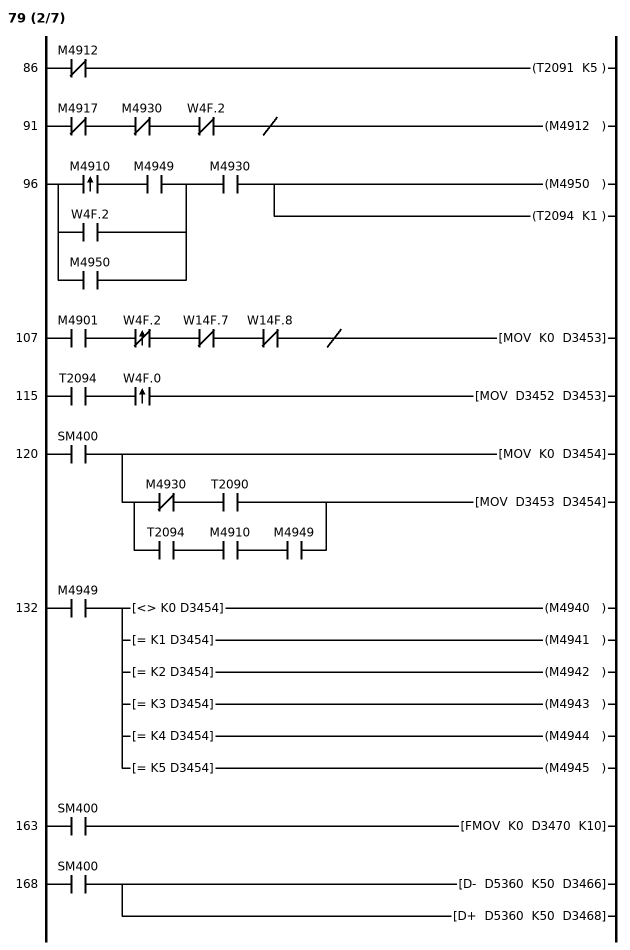
86    LDI     M4912
      OUT     T2091 K5
91    LDI     M4917
      ANI     M4930
      ANI     W4F.2
      INV
      OUT     M4912
96    LDP     M4910
      AND     M4949
      OR      W4F.2
      OR      M4950
      AND     M4930
      OUT     M4950
      OUT     T2094 K1
107   LD      M4901
      ANDPI   W4F.2
      ANI     W14F.7
      ANI     W14F.8
      INV
      MOV     K0 D3453
115   LD      T2094
      ANDP    W4F.0
      MOV     D3452 D3453
120   LD      SM400
      MOV     K0 D3454
      LDI     M4930
      AND     T2090
      LD      T2094
      AND     M4910
      AND     M4949
      ORB
      ANB
      MOV     D3453 D3454
132   LD      M4949
      MPS
      AND<>   K0 D3454
      OUT     M4940
      MRD
      AND=    K1 D3454
      OUT     M4941
      MRD
      AND=    K2 D3454
      OUT     M4942
      MRD
      AND=    K3 D3454
      OUT     M4943
      MRD
      AND=    K4 D3454
      OUT     M4944
      MPP
      AND=    K5 D3454
      OUT     M4945
163   LD      SM400
      FMOV    K0 D3470 K10
168   LD      SM400
      D-      D5360 K50 D3466
      D+      D5360 K50 D3468
